// TIA Portal project "Elevator" (V15)

(* hardware
DEVICE "S7300/ET200M station_1"  S7-300 station
   slot 0: "Rail_0"  Rail  6ES7 390-1***0-0AA0
   slot 2: "PLC_1"  CPU 313C-2 DP  6ES7 313-6CF03-0AB0  V2.6
      slot 0: "MPI interface_1"  X1
      slot 1: "DP interface_1"  X2
      slot 2: "DI 16/DO 16_1"  DI16/DO16
      slot 4: "Count_1"  Counter
*)

// ===== PLC "PLC_1"  CPU 313C-2 DP =====

VAR_GLOBAL   // PLC tag table "Default tag table"
   "Encoder" AT %I0.0 : Bool;
   "house" AT %I0.3 : Bool;
   "motorup" AT %Q0.3 : Bool;
   "motordown" AT %Q0.1 : Bool;
   "Flat" AT %MW10 : Int;
   "Currentflat" AT %MW12 : Int;
   "Start" AT %M0.0 : Bool;
   "Stop" AT %M0.1 : Bool;
   "Pulses" AT %MD30 : DInt;
   "Reset" AT %M0.2 : Bool;
   "Pulses_Req" AT %MD14 : DInt;
   "temp" AT %MW20 : Int;
   "OK" AT %M0.3 : Bool;
   "f1" AT %MW24 : Int;
   "f2" AT %MD40 : DInt;
   "f3" AT %M0.4 : Bool;
   "f4" AT %M0.5 : Bool;
   "f5" AT %M0.6 : Bool;
   "i0" AT %M50.0 : Bool;
   "i1" AT %M50.1 : Bool;
   "i2" AT %M50.2 : Bool;
   "i3" AT %M50.3 : Bool;
   "i4" AT %M50.4 : Bool;
   "i5" AT %M50.5 : Bool;
   "o0" AT %M50.6 : Bool;
   "o1" AT %M50.7 : Bool;
   "o2" AT %M51.0 : Bool;
   "o3" AT %M51.1 : Bool;
   "o4" AT %M51.2 : Bool;
   "o5" AT %M51.3 : Bool;
   "marker up" AT %M51.4 : Bool;
   "marker down" AT %M51.5 : Bool;
END_VAR

FUNCTION "main code" : Void   // FC1, SCL
{ S7_Optimized_Access := 'FALSE' }
VERSION : 0.1
BEGIN
   REGION Up OR Dn
       IF "f5" = 1 THEN
           IF "Flat" < "Currentflat" THEN
               "motordown" := 1;
           END_IF;

           IF "Flat" > "Currentflat" THEN
               "motorup" := 1;
           END_IF;
       END_IF;
   END_REGION

   REGION Compare encoder
     IF "motorup" = 1 THEN
           "marker up" := 1;
       END_IF;
     IF "motordown" THEN
           "marker up" := 0;
       END_IF;

       IF "marker up" = 1 THEN

           IF "o5" = 1 THEN
               "Flat" := 5;
           ELSIF "o4" = 1 THEN
               "Flat" := 4;
           ELSIF "o3" = 1 THEN
               "Flat" := 3;
           ELSIF "o2" = 1 THEN
               "Flat" := 2;
           ELSIF "o1" = 1 THEN
               "Flat" := 1;
           ELSIF "o0" = 1 THEN
               "Flat" := 0;
           END_IF;

           IF "i0" = 1 THEN
               "Flat" := 0;
           ELSIF "i1" = 1 THEN
               "Flat" := 1;
           ELSIF "i2" = 1 THEN
               "Flat" := 2;
           ELSIF "i3" = 1 THEN
               "Flat" := 3;
           ELSIF "i4" = 1 THEN
               "Flat" := 4;
           ELSIF "i5" = 1 THEN
               "Flat" := 5;
           END_IF;

      END_IF;

       IF "marker up" = 0 THEN

           IF "i5" = 1 OR "o5" = 1 THEN
               "Flat" := 5;
           ELSIF "i4" = 1 OR "o4" = 1 THEN
               "Flat" := 4;
           ELSIF "i3" = 1 OR "o3" = 1 THEN
               "Flat" := 3;
           ELSIF "i2" = 1 OR "o2" = 1 THEN
               "Flat" := 2;
           ELSIF "i1" = 1 OR "o1" = 1 THEN
               "Flat" := 1;
           ELSIF "i0" = 1 OR "o0" = 1 THEN
               "Flat" := 0;
           END_IF;

       END_IF;


   END_REGION

   REGION Reset Markers
       IF "motordown" = 0 AND "motorup" = 0 THEN
           IF "Currentflat" = 5 THEN
               "i5" := 0;
               "o5" := 0;
           END_IF;
           IF "Currentflat" = 4 THEN
               "i4" := 0;
               "o4" := 0;
           END_IF;
           IF "Currentflat" = 3 THEN
               "i3" := 0;
               "o3" := 0;
           END_IF;
           IF "Currentflat" = 2 THEN
               "i2" := 0;
               "o2" := 0;
           END_IF;
           IF "Currentflat" = 1 THEN
               "i1" := 0;
               "o1" := 0;
           END_IF;
           IF "Currentflat" = 0 THEN
               "i0" := 0;
               "o0" := 0;
           END_IF;
       END_IF; 
   END_REGION

   REGION Compare encoder

       "f1" := "Flat" - "Currentflat";
       "f1" := "f1" * 150;
       "f2" := INT_TO_DINT("f1");
       "f2" := ABS_DINT("f2");

       IF "f2" - "Pulses" = 0 THEN
           "motordown" := 0;
           "motorup" := 0;
           "Currentflat" := "Flat";

       END_IF;


   END_REGION
END_FUNCTION

ORGANIZATION_BLOCK "Main"   // OB1, LAD
TITLE = "Main Program Sweep (Cycle)"
{ S7_Optimized_Access := 'FALSE' }
VERSION : 0.1
   VAR_TEMP
      OB1_EV_CLASS : Byte;   // Bits 0-3 = 1 (Coming event), Bits 4-7 = 1 (Event class 1)
      OB1_SCAN_1 : Byte;   // 1 (Cold restart scan 1 of OB 1), 3 (Scan 2-n of OB 1)
      OB1_PRIORITY : Byte;   // Priority of OB Execution
      OB1_OB_NUMBR : Byte;   // 1 (Organization block 1, OB1)
      OB1_RESERVED_1 : Byte;   // Reserved for system
      OB1_RESERVED_2 : Byte;   // Reserved for system
      OB1_PREV_CYCLE : Int;   // Cycle time of previous OB1 scan (milliseconds)
      OB1_MIN_CYCLE : Int;   // Minimum cycle time of OB1 (milliseconds)
      OB1_MAX_CYCLE : Int;   // Maximum cycle time of OB1 (milliseconds)
      OB1_DATE_TIME : Date_And_Time;   // Date and time OB1 started
   END_VAR
   VAR_TEMP   // added for the SCL form of the ladder/FBD networks
      _w1 : Bool;
   END_VAR
BEGIN

REGION Network 1
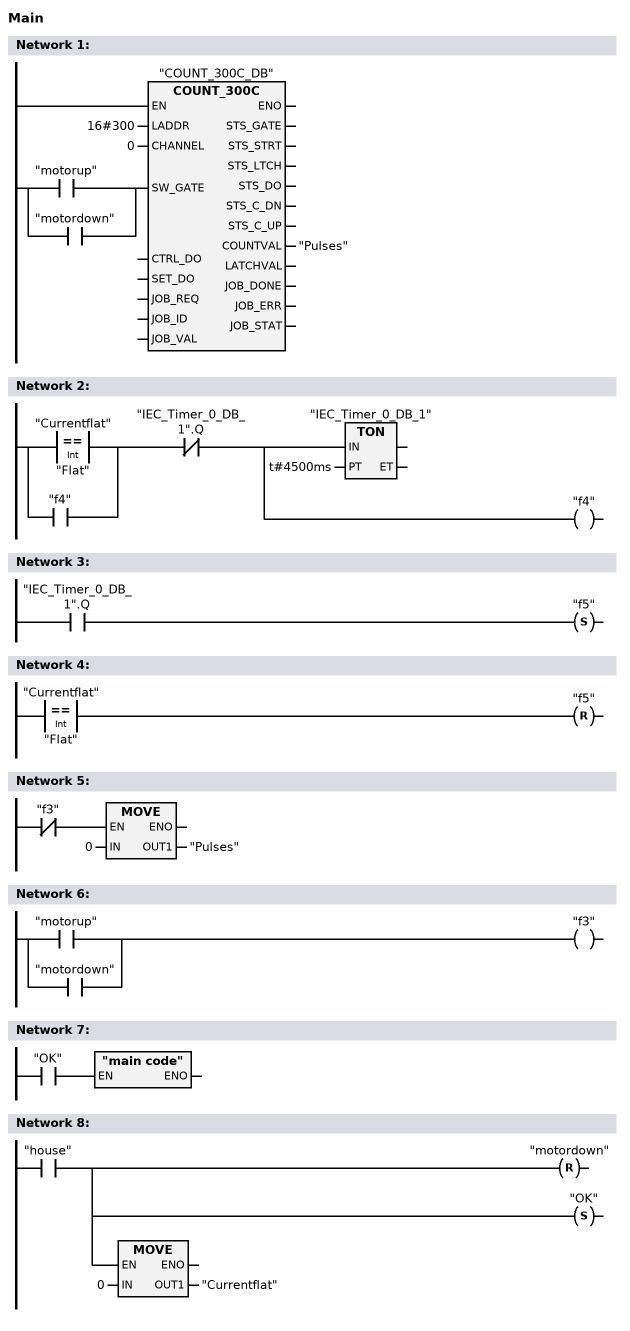
   "COUNT_300C_DB"(LADDR := 16#300, CHANNEL := 0, SW_GATE := "motorup" OR "motordown", COUNTVAL => "Pulses");   // COUNT_300C
END_REGION

REGION Network 2
   #_w1 := (("Currentflat" = "Flat") OR "f4") AND NOT "IEC_Timer_0_DB_1".Q;
   "IEC_Timer_0_DB_1".TON(IN := #_w1, PT := t#4500ms);
   "f4" := #_w1;
END_REGION

REGION Network 3
   RUNG wire#powerrail
      Contact( "IEC_Timer_0_DB_1".Q )
      S_Coil( "f5" )
   END_RUNG
   // the same network as SCL:
   IF "IEC_Timer_0_DB_1".Q THEN "f5" := TRUE; END_IF;
END_REGION

REGION Network 4
   RUNG wire#powerrail
      { S7_Templates := "SrcType := Int" } EQ_Contact(in1 := "Currentflat", in2 := "Flat")
      R_Coil( "f5" )
   END_RUNG
   // the same network as SCL:
   IF "Currentflat" = "Flat" THEN "f5" := FALSE; END_IF;
END_REGION

REGION Network 5
   RUNG wire#powerrail
      I_Contact( "f3" )
      { S7_GenerateENO := "TRUE" } Move(in := 0, out1 => "Pulses")
   END_RUNG
   // the same network as SCL:
   IF NOT "f3" THEN "Pulses" := 0; END_IF;
END_REGION

REGION Network 6
   RUNG wire#powerrail
      Contact( "motorup" )
      wire#w1
      Coil( "f3" )
   END_RUNG
   RUNG wire#powerrail
      Contact( "motordown" )
   END_RUNG wire#w1
   // the same network as SCL:
   "f3" := "motorup" OR "motordown";
END_REGION

REGION Network 7
   RUNG wire#powerrail
      Contact( "OK" )
      "main code"()
   END_RUNG
   // the same network as SCL:
   IF "OK" THEN "main code"(); END_IF;
END_REGION

REGION Network 8
   RUNG wire#powerrail
      Contact( "house" )
      wire#w1
      R_Coil( "motordown" )
   END_RUNG
   RUNG wire#w1
      S_Coil( "OK" )
   END_RUNG
   RUNG wire#w1
      { S7_GenerateENO := "TRUE" } Move(in := 0, out1 => "Currentflat")
   END_RUNG
   // the same network as SCL:
   IF "house" THEN
       "motordown" := FALSE;
       "OK" := TRUE;
       "Currentflat" := 0;
   END_IF;
END_REGION
END_ORGANIZATION_BLOCK

ORGANIZATION_BLOCK "COMM_FLT"   // OB87, LAD
TITLE = "Communication Fault"
{ S7_Optimized_Access := 'FALSE' }
VERSION : 0.1
   VAR_TEMP
      OB87_EV_CLASS : Byte;   // 16#39 Event class 3
      OB87_FLT_ID : Byte;   // 16#XX, Fault identifcation code
      OB87_PRIORITY : Byte;   // Priority of OB Execution
      OB87_OB_NUMBR : Byte;   // 87 (Organization block 87, OB87)
      OB87_RESERVED_1 : Byte;   // Reserved for system
      OB87_RESERVED_2 : Byte;   // Reserved for system
      OB87_RESERVED_3 : Word;   // Reserved for system
      OB87_RESERVED_4 : DWord;   // Reserved for system
      OB87_DATE_TIME : Date_And_Time;   // Date and time OB87 started
   END_VAR
BEGIN
END_ORGANIZATION_BLOCK

ORGANIZATION_BLOCK "Startup"   // OB100, SCL
TITLE = "Complete Restart"
{ S7_Optimized_Access := 'FALSE' }
VERSION : 0.1
   VAR_TEMP
      OB100_EV_CLASS : Byte;   // 16#13, Event class 1, Entering event state, Event logged in diagnostic buffer
      OB100_STRTUP : Byte;   // 16#81/82/83/84 Method of startup
      OB100_PRIORITY : Byte;   // Priority of OB Execution
      OB100_OB_NUMBR : Byte;   // 100 (Organization block 100, OB100)
      OB100_RESERVED_1 : Byte;   // Reserved for system
      OB100_RESERVED_2 : Byte;   // Reserved for system
      OB100_STOP : Word;   // Event that caused CPU to stop (16#4xxx)
      OB100_STRT_INFO : DWord;   // Information on how system started
      OB100_DATE_TIME : Date_And_Time;   // Date and time OB100 started
   END_VAR
BEGIN
   "motordown" := 1;
END_ORGANIZATION_BLOCK

ORGANIZATION_BLOCK "PROG_ERR"   // OB121, LAD
TITLE = "Programming Error"
{ S7_Optimized_Access := 'FALSE' }
VERSION : 0.1
   VAR_TEMP
      OB121_EV_CLASS : Byte;   // 16#25, Event class 2, Entering event state, Internal fault event
      OB121_SW_FLT : Byte;   // 16#XX Software programming fault
      OB121_PRIORITY : Byte;   // Priority of OB Execution
      OB121_OB_NUMBR : Byte;   // 121 (Organization block 121, OB121)
      OB121_BLK_TYPE : Byte;   // 16#88/8A/8B/8C/8E Type of block fault occured in
      OB121_RESERVED_1 : Byte;   // Reserved for system
      OB121_FLT_REG : Word;   // 16#XX Specific register that caused fault
      OB121_BLK_NUM : Word;   // Number of block that programming fault occured in
      OB121_PRG_ADDR : Word;   // Address in block where programming fault occured
      OB121_DATE_TIME : Date_And_Time;   // Date and time OB121 started
   END_VAR
BEGIN
END_ORGANIZATION_BLOCK